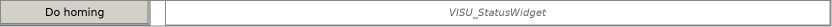
VISUALIZATION VISU_Axes_Commands_DoHoming  // 832x27
VAR_IN_OUT
    doHoming : AxesDoHomingProcess;
    doHomingStatus : StatusWidget;
END_VAR
    Button (0,0 150x25), "Do homing", input disabled if: doHoming.statuses.enabledStatus.disabled
        OnMouseClick: execute { doHoming.request(); }
    Frame (165,0 665x25)
        shows VISU_StatusWidget(widget := doHomingStatus)
END_VISUALIZATION

(* stored: Version 1.1.0.1, ProductVersion 3.1.4019.2
   Visu VISU_Axes_Commands_DoHoming: Id {f75008ed-618c-4e2b-ad13-9ab9246038a7} *)
